{attribute 'GeneratedUsingTerminal: EL9210-0000-0016'}
{attribute addProperty BoxType "EL9210-0000-0016"}
{attribute addProperty Id "PowerOKAT %I*PowerOK_CEB2FD121FuseErrorAT %I*FuseError_1EC650DA1WcStateAT %I*WcState_9091E0EB2InfoDataAT %I*InfoData_6F19DB2B2"}
{attribute addProperty CRC "3015756419"}
{attribute addProperty Size "6"}
TYPE EL9210_B3C0CA83 :
STRUCT
	{attribute addProperty Name "PowerOK"}
	PowerOK : PowerOK_CEB2FD12;
	{attribute addProperty Name "FuseError"}
	FuseError : FuseError_1EC650DA;
	{attribute addProperty Name "WcState"}
	WcState : WcState_9091E0EB;
	{attribute addProperty Name "InfoData"}
	InfoData : InfoData_6F19DB2B;
END_STRUCT
END_TYPE

(* stored: Version 1.2.0.0, ProductVersion 3.1.4024.9
   DUT EL9210_B3C0CA83: Id {069f6d0f-e6fd-4d21-ae2c-8a10f1d6837b} *)
